PROGRAM P00_Mapping
VAR
	AI_SPARE								:INT;
	DI_SPARE								:BOOL;
	AO_SPARE								:INT:=0;
	DO_SPARE								:BOOL:=FALSE;
	
	
	TI1										:ST_EL3214;
	AI1										:ST_EL3174;
	AI2										:ST_EL3174;
	DI1										:ST_EL1819;
	AO1										:ST_EL4124;
	PS1										:ST_EL9110;
	DO1										:ST_EL2809;
	DO2										:ST_EL2809;
	PB1										:ST_EL6021;


END_VAR

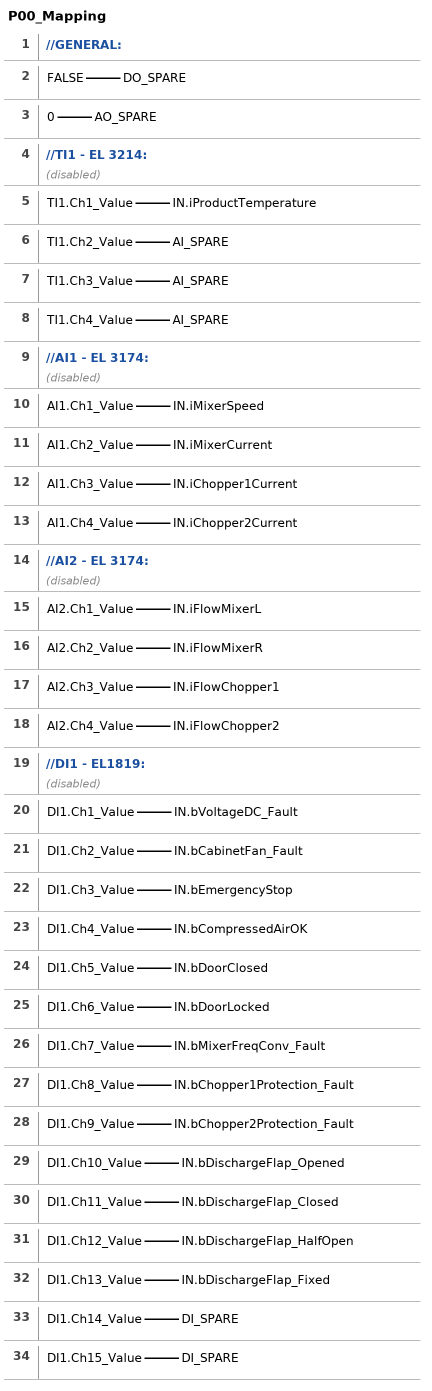
// NETWORK 1
// label: //GENERAL

// NETWORK 2
DO_SPARE := FALSE;

// NETWORK 3
AO_SPARE := 0;

// NETWORK 4 (disabled)
// label: //TI1 - EL 3214

// NETWORK 5
IN.iProductTemperature := TI1.Ch1_Value;

// NETWORK 6
AI_SPARE := TI1.Ch2_Value;

// NETWORK 7
AI_SPARE := TI1.Ch3_Value;

// NETWORK 8
AI_SPARE := TI1.Ch4_Value;

// NETWORK 9 (disabled)
// label: //AI1 - EL 3174

// NETWORK 10
IN.iMixerSpeed := AI1.Ch1_Value;

// NETWORK 11
IN.iMixerCurrent := AI1.Ch2_Value;

// NETWORK 12
IN.iChopper1Current := AI1.Ch3_Value;

// NETWORK 13
IN.iChopper2Current := AI1.Ch4_Value;

// NETWORK 14 (disabled)
// label: //AI2 - EL 3174

// NETWORK 15
IN.iFlowMixerL := AI2.Ch1_Value;

// NETWORK 16
IN.iFlowMixerR := AI2.Ch2_Value;

// NETWORK 17
IN.iFlowChopper1 := AI2.Ch3_Value;

// NETWORK 18
IN.iFlowChopper2 := AI2.Ch4_Value;

// NETWORK 19 (disabled)
// label: //DI1 - EL1819

// NETWORK 20
IN.bVoltageDC_Fault := DI1.Ch1_Value;

// NETWORK 21
IN.bCabinetFan_Fault := DI1.Ch2_Value;

// NETWORK 22
IN.bEmergencyStop := DI1.Ch3_Value;

// NETWORK 23
IN.bCompressedAirOK := DI1.Ch4_Value;

// NETWORK 24
IN.bDoorClosed := DI1.Ch5_Value;

// NETWORK 25
IN.bDoorLocked := DI1.Ch6_Value;

// NETWORK 26
IN.bMixerFreqConv_Fault := DI1.Ch7_Value;

// NETWORK 27
IN.bChopper1Protection_Fault := DI1.Ch8_Value;

// NETWORK 28
IN.bChopper2Protection_Fault := DI1.Ch9_Value;

// NETWORK 29
IN.bDischargeFlap_Opened := DI1.Ch10_Value;

// NETWORK 30
IN.bDischargeFlap_Closed := DI1.Ch11_Value;

// NETWORK 31
IN.bDischargeFlap_HalfOpen := DI1.Ch12_Value;

// NETWORK 32
IN.bDischargeFlap_Fixed := DI1.Ch13_Value;

// NETWORK 33
DI_SPARE := DI1.Ch14_Value;

// NETWORK 34
DI_SPARE := DI1.Ch15_Value;

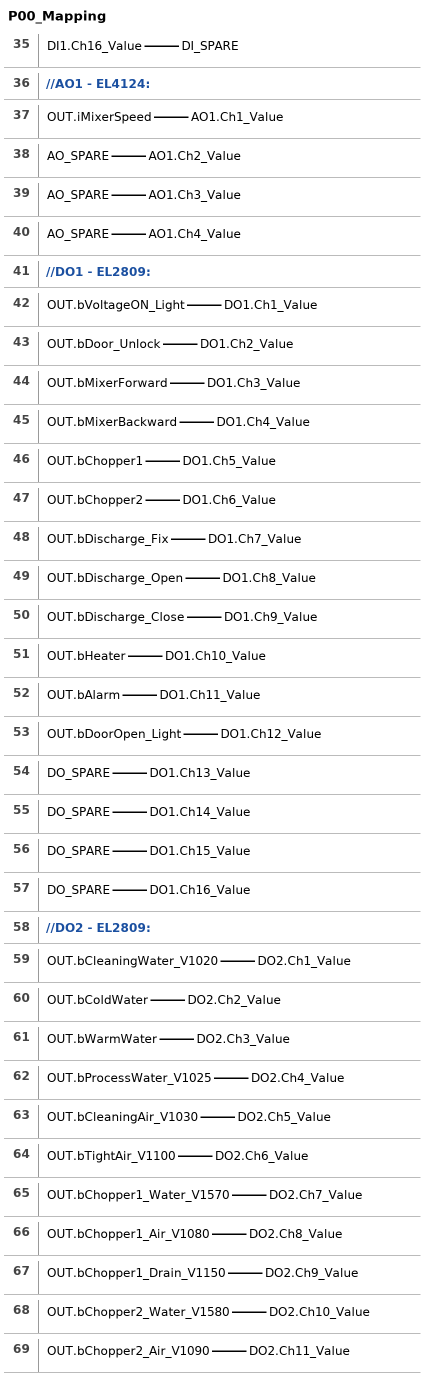
// NETWORK 35
DI_SPARE := DI1.Ch16_Value;

// NETWORK 36
// label: //AO1 - EL4124

// NETWORK 37
AO1.Ch1_Value := OUT.iMixerSpeed;

// NETWORK 38
AO1.Ch2_Value := AO_SPARE;

// NETWORK 39
AO1.Ch3_Value := AO_SPARE;

// NETWORK 40
AO1.Ch4_Value := AO_SPARE;

// NETWORK 41
// label: //DO1 - EL2809

// NETWORK 42
DO1.Ch1_Value := OUT.bVoltageON_Light;

// NETWORK 43
DO1.Ch2_Value := OUT.bDoor_Unlock;

// NETWORK 44
DO1.Ch3_Value := OUT.bMixerForward;

// NETWORK 45
DO1.Ch4_Value := OUT.bMixerBackward;

// NETWORK 46
DO1.Ch5_Value := OUT.bChopper1;

// NETWORK 47
DO1.Ch6_Value := OUT.bChopper2;

// NETWORK 48
DO1.Ch7_Value := OUT.bDischarge_Fix;

// NETWORK 49
DO1.Ch8_Value := OUT.bDischarge_Open;

// NETWORK 50
DO1.Ch9_Value := OUT.bDischarge_Close;

// NETWORK 51
DO1.Ch10_Value := OUT.bHeater;

// NETWORK 52
DO1.Ch11_Value := OUT.bAlarm;

// NETWORK 53
DO1.Ch12_Value := OUT.bDoorOpen_Light;

// NETWORK 54
DO1.Ch13_Value := DO_SPARE;

// NETWORK 55
DO1.Ch14_Value := DO_SPARE;

// NETWORK 56
DO1.Ch15_Value := DO_SPARE;

// NETWORK 57
DO1.Ch16_Value := DO_SPARE;

// NETWORK 58
// label: //DO2 - EL2809

// NETWORK 59
DO2.Ch1_Value := OUT.bCleaningWater_V1020;

// NETWORK 60
DO2.Ch2_Value := OUT.bColdWater;

// NETWORK 61
DO2.Ch3_Value := OUT.bWarmWater;

// NETWORK 62
DO2.Ch4_Value := OUT.bProcessWater_V1025;

// NETWORK 63
DO2.Ch5_Value := OUT.bCleaningAir_V1030;

// NETWORK 64
DO2.Ch6_Value := OUT.bTightAir_V1100;

// NETWORK 65
DO2.Ch7_Value := OUT.bChopper1_Water_V1570;

// NETWORK 66
DO2.Ch8_Value := OUT.bChopper1_Air_V1080;

// NETWORK 67
DO2.Ch9_Value := OUT.bChopper1_Drain_V1150;

// NETWORK 68
DO2.Ch10_Value := OUT.bChopper2_Water_V1580;

// NETWORK 69
DO2.Ch11_Value := OUT.bChopper2_Air_V1090;

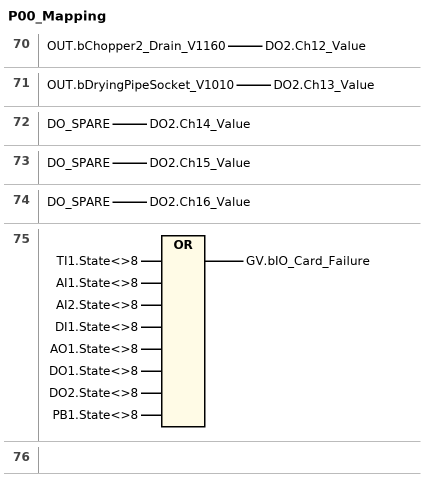
// NETWORK 70
DO2.Ch12_Value := OUT.bChopper2_Drain_V1160;

// NETWORK 71
DO2.Ch13_Value := OUT.bDryingPipeSocket_V1010;

// NETWORK 72
DO2.Ch14_Value := DO_SPARE;

// NETWORK 73
DO2.Ch15_Value := DO_SPARE;

// NETWORK 74
DO2.Ch16_Value := DO_SPARE;

// NETWORK 75
GV.bIO_Card_Failure := (TI1.State<>8) OR (AI1.State<>8) OR (AI2.State<>8) OR (DI1.State<>8) OR (AO1.State<>8) OR (DO1.State<>8) OR (DO2.State<>8) OR (PB1.State<>8);

// NETWORK 76

END_PROGRAM

(* stored: Version 1.1.0.1
   POU P00_Mapping: Id {98a147a1-4723-4394-a592-65dcb4825381}, SpecialFunc None *)
